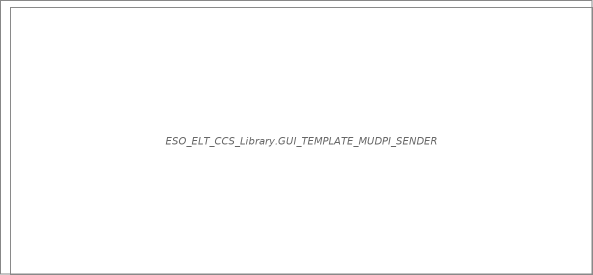
VISUALIZATION GUI_MUDPI_SENDER  // 593x275
    Frame (10,7 583x268)
        shows ESO_ELT_CCS_Library.GUI_TEMPLATE_MUDPI_SENDER(m_Instance := MAIN.fbSender)
END_VISUALIZATION

(* stored: Version 1.1.0.1, ProductVersion 3.1.4024.9
   Visu GUI_MUDPI_SENDER: Id {efff83ac-22c4-4fc0-85fc-b3f98d8ba69a} *)
